// LS Electric XG5000 project: R11_plc
// PLC LoadWizard_PLC
// module base 0 slot 0: FEnet:XGL-EFMT(B) (Fast Ethernet Module, Electrical Master)
// module base 0 slot 1: Input Module:XGI-D24A/B (DC 24V Input, 32 Contacts)
// module base 0 slot 2: Output Module:XGQ-TR4A/B (Transistor Output, 32 Contacts (0.1A, Sink Output/Source Output))
// module base 0 slot 3: 64points reservation:XG-IN64

PROGRAM Main (task: Scan Program)

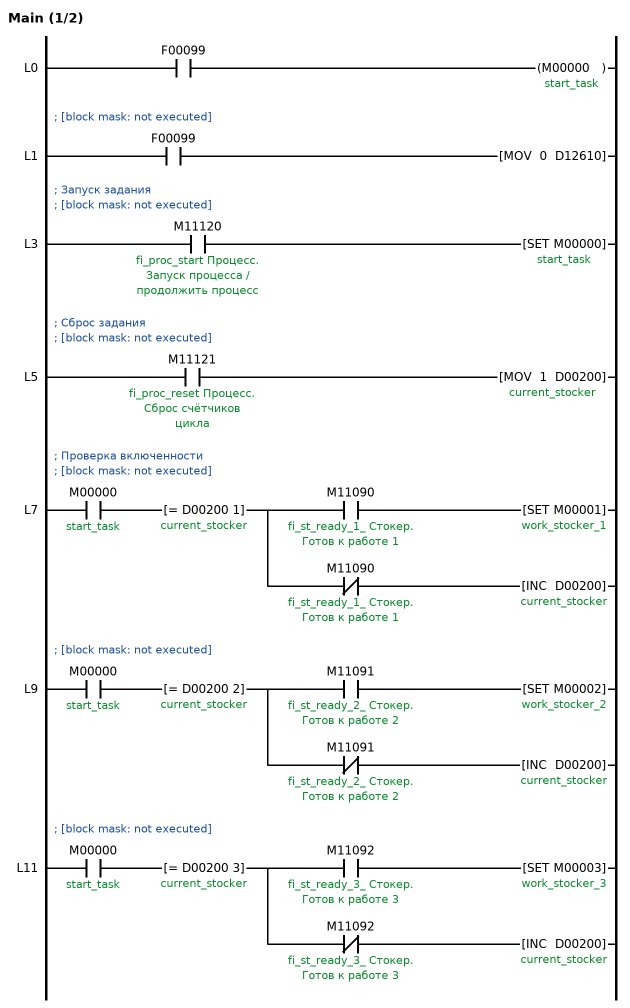
; L0
LOAD      F00099
OUT       M00000	// start_task
; L1 (block mask: not executed)
LOAD      F00099
MOV       0 D12610
// Запуск задания
; L3 (block mask: not executed)
LOAD      M11120	// fi_proc_start Процесс. Запуск процесса / продолжить процесс
SET       M00000	// start_task
// Сброс задания
; L5 (block mask: not executed)
LOAD      M11121	// fi_proc_reset Процесс. Сброс счётчиков цикла
MOV       1 D00200	// current_stocker
// Проверка включенности
; L7 (block mask: not executed)
LOAD      M00000	// start_task
AND=      D00200 1	// current_stocker
MPUSH
AND       M11090	// fi_st_ready_1_ Стокер. Готов к работе 1
SET       M00001	// work_stocker_1
MPOP
AND NOT   M11090	// fi_st_ready_1_ Стокер. Готов к работе 1
INC       D00200	// current_stocker
; L9 (block mask: not executed)
LOAD      M00000	// start_task
AND=      D00200 2	// current_stocker
MPUSH
AND       M11091	// fi_st_ready_2_ Стокер. Готов к работе 2
SET       M00002	// work_stocker_2
MPOP
AND NOT   M11091	// fi_st_ready_2_ Стокер. Готов к работе 2
INC       D00200	// current_stocker
; L11 (block mask: not executed)
LOAD      M00000	// start_task
AND=      D00200 3	// current_stocker
MPUSH
AND       M11092	// fi_st_ready_3_ Стокер. Готов к работе 3
SET       M00003	// work_stocker_3
MPOP
AND NOT   M11092	// fi_st_ready_3_ Стокер. Готов к работе 3
INC       D00200	// current_stocker

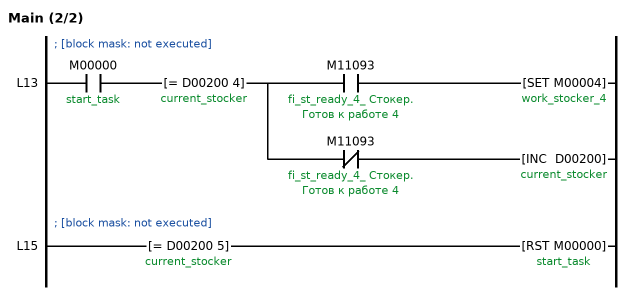
; L13 (block mask: not executed)
LOAD      M00000	// start_task
AND=      D00200 4	// current_stocker
MPUSH
AND       M11093	// fi_st_ready_4_ Стокер. Готов к работе 4
SET       M00004	// work_stocker_4
MPOP
AND NOT   M11093	// fi_st_ready_4_ Стокер. Готов к работе 4
INC       D00200	// current_stocker
; L15 (block mask: not executed)
LOAD=     D00200 5	// current_stocker
RST       M00000	// start_task

PROGRAM CNC (task: Scan Program)

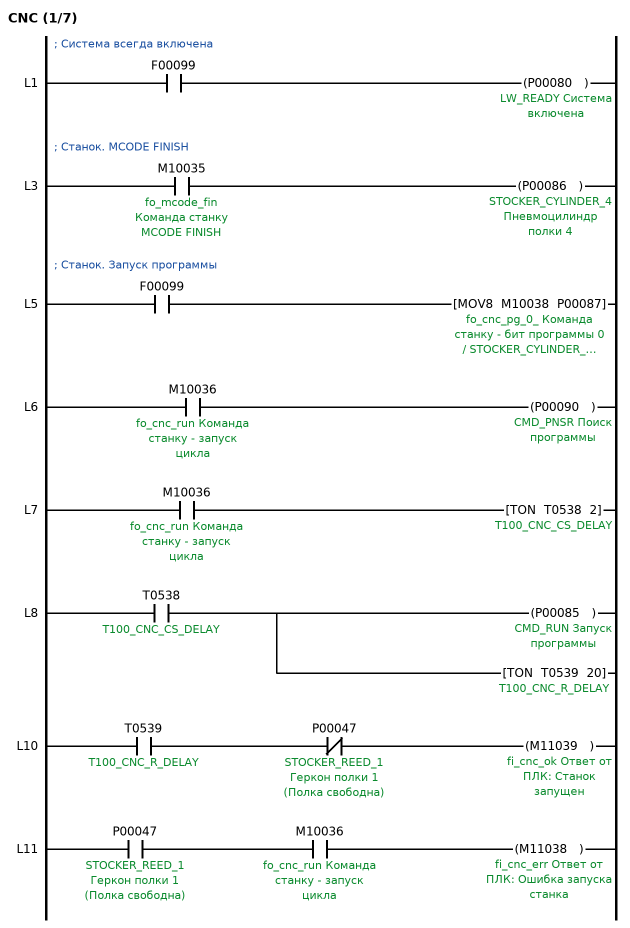
// Система всегда включена
; L1
LOAD      F00099
OUT       P00080	// LW_READY Система включена
// Станок. MCODE FINISH
; L3
LOAD      M10035	// fo_mcode_fin Команда станку  MCODE FINISH
OUT       P00086	// STOCKER_CYLINDER_4 Пневмоцилиндр полки 4
// Станок. Запуск программы
; L5
LOAD      F00099
MOV8      M10038 P00087	// fo_cnc_pg_0_ Команда станку - бит программы 0 / STOCKER_CYLINDER_3 Пневмоцилиндр полки 3
; L6
LOAD      M10036	// fo_cnc_run Команда станку - запуск цикла
OUT       P00090	// CMD_PNSR Поиск программы
; L7
LOAD      M10036	// fo_cnc_run Команда станку - запуск цикла
TON       T0538 2	// T100_CNC_CS_DELAY
; L8
LOAD      T0538	// T100_CNC_CS_DELAY
OUT       P00085	// CMD_RUN Запуск программы
TON       T0539 20	// T100_CNC_R_DELAY
; L10
LOAD      T0539	// T100_CNC_R_DELAY
AND NOT   P00047	// STOCKER_REED_1 Геркон полки 1 (Полка свободна)
OUT       M11039	// fi_cnc_ok Ответ от ПЛК: Станок запущен 
; L11
LOAD      P00047	// STOCKER_REED_1 Геркон полки 1 (Полка свободна)
AND       M10036	// fo_cnc_run Команда станку - запуск цикла
OUT       M11038	// fi_cnc_err Ответ от ПЛК: Ошибка запуска станка

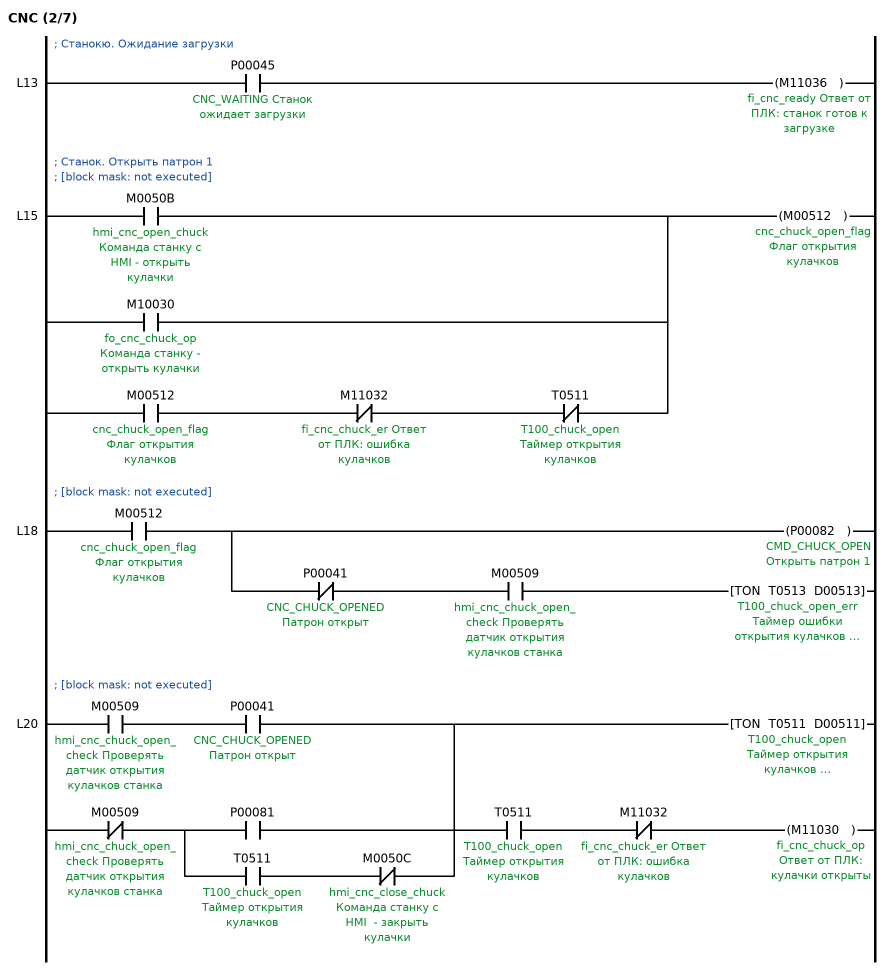
// Станокю. Ожидание загрузки
; L13
LOAD      P00045	// CNC_WAITING Станок ожидает загрузки
OUT       M11036	// fi_cnc_ready Ответ от ПЛК: станок готов к загрузке
// Станок. Открыть патрон 1
; L15 (block mask: not executed)
LOAD      M0050B	// hmi_cnc_open_chuck Команда станку с HMI - открыть кулачки
OR        M10030	// fo_cnc_chuck_op Команда станку - открыть кулачки
LOAD      M00512	// cnc_chuck_open_flag Флаг открытия кулачков
AND NOT   M11032	// fi_cnc_chuck_er Ответ от ПЛК: ошибка кулачков
AND NOT   T0511	// T100_chuck_open Таймер открытия кулачков
OR LOAD
OUT       M00512	// cnc_chuck_open_flag Флаг открытия кулачков
; L18 (block mask: not executed)
LOAD      M00512	// cnc_chuck_open_flag Флаг открытия кулачков
OUT       P00082	// CMD_CHUCK_OPEN Открыть патрон 1
AND NOT   P00041	// CNC_CHUCK_OPENED Патрон открыт
AND       M00509	// hmi_cnc_chuck_open_check Проверять датчик открытия кулачков станка
TON       T0513 D00513	// T100_chuck_open_err Таймер ошибки открытия кулачков / hmi_chuck_err_time Время ошибки кулачков
; L20 (block mask: not executed)
LOAD      M00509	// hmi_cnc_chuck_open_check Проверять датчик открытия кулачков станка
AND       P00041	// CNC_CHUCK_OPENED Патрон открыт
LOAD NOT  M00509	// hmi_cnc_chuck_open_check Проверять датчик открытия кулачков станка
LOAD      P00081
LOAD      T0511	// T100_chuck_open Таймер открытия кулачков
AND NOT   M0050C	// hmi_cnc_close_chuck Команда станку с HMI  - закрыть кулачки
OR LOAD
AND LOAD
OR LOAD
TON       T0511 D00511	// T100_chuck_open Таймер открытия кулачков / hmi_chuck_open_time Время на открытие кулачков
AND       T0511	// T100_chuck_open Таймер открытия кулачков
AND NOT   M11032	// fi_cnc_chuck_er Ответ от ПЛК: ошибка кулачков
OUT       M11030	// fi_cnc_chuck_op Ответ от ПЛК: кулачки открыты

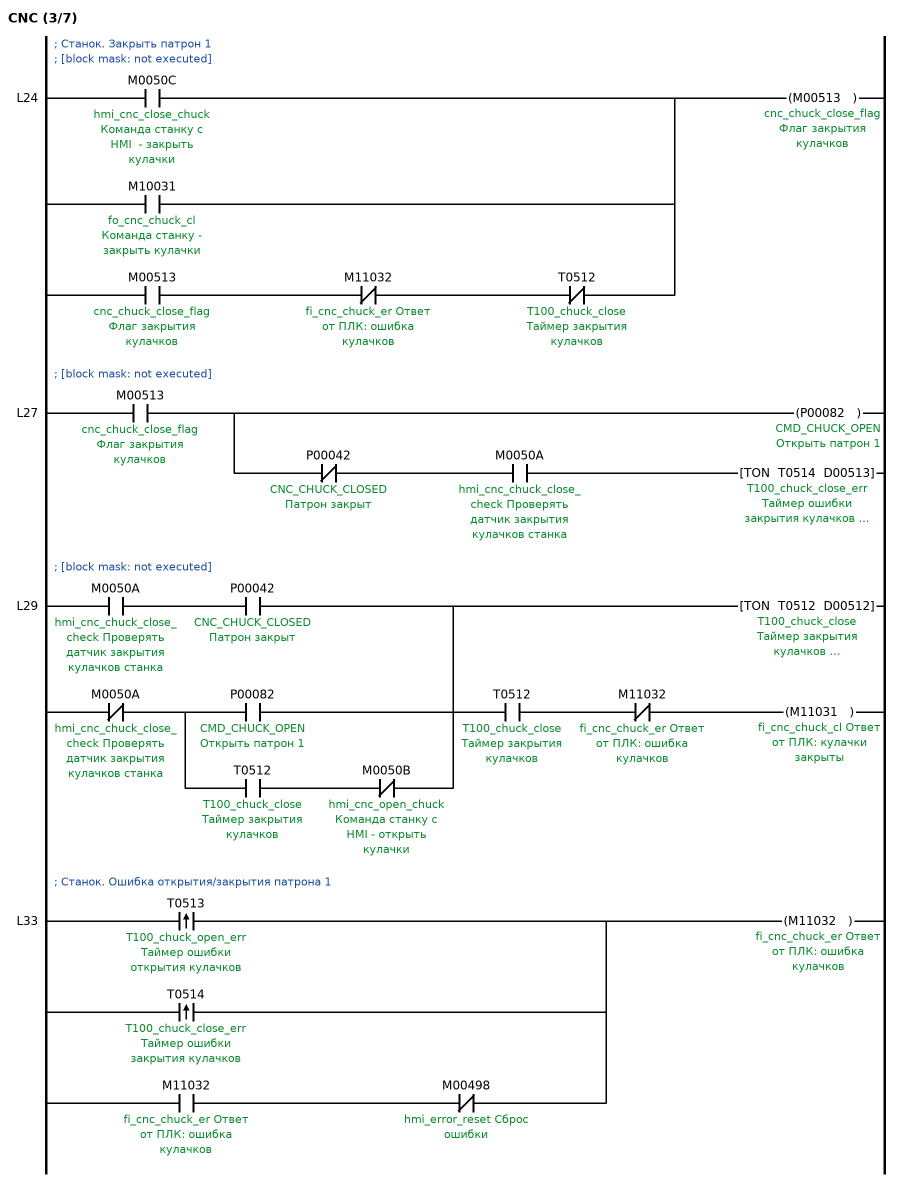
// Станок. Закрыть патрон 1
; L24 (block mask: not executed)
LOAD      M0050C	// hmi_cnc_close_chuck Команда станку с HMI  - закрыть кулачки
OR        M10031	// fo_cnc_chuck_cl Команда станку - закрыть кулачки
LOAD      M00513	// cnc_chuck_close_flag Флаг закрытия кулачков
AND NOT   M11032	// fi_cnc_chuck_er Ответ от ПЛК: ошибка кулачков
AND NOT   T0512	// T100_chuck_close Таймер закрытия кулачков
OR LOAD
OUT       M00513	// cnc_chuck_close_flag Флаг закрытия кулачков
; L27 (block mask: not executed)
LOAD      M00513	// cnc_chuck_close_flag Флаг закрытия кулачков
OUT       P00082	// CMD_CHUCK_OPEN Открыть патрон 1
AND NOT   P00042	// CNC_CHUCK_CLOSED Патрон закрыт
AND       M0050A	// hmi_cnc_chuck_close_check Проверять датчик закрытия кулачков станка
TON       T0514 D00513	// T100_chuck_close_err Таймер ошибки закрытия кулачков / hmi_chuck_err_time Время ошибки кулачков
; L29 (block mask: not executed)
LOAD      M0050A	// hmi_cnc_chuck_close_check Проверять датчик закрытия кулачков станка
AND       P00042	// CNC_CHUCK_CLOSED Патрон закрыт
LOAD NOT  M0050A	// hmi_cnc_chuck_close_check Проверять датчик закрытия кулачков станка
LOAD      P00082	// CMD_CHUCK_OPEN Открыть патрон 1
LOAD      T0512	// T100_chuck_close Таймер закрытия кулачков
AND NOT   M0050B	// hmi_cnc_open_chuck Команда станку с HMI - открыть кулачки
OR LOAD
AND LOAD
OR LOAD
TON       T0512 D00512	// T100_chuck_close Таймер закрытия кулачков / hmi_chuck_close_time Время на закрытие кулачков
AND       T0512	// T100_chuck_close Таймер закрытия кулачков
AND NOT   M11032	// fi_cnc_chuck_er Ответ от ПЛК: ошибка кулачков
OUT       M11031	// fi_cnc_chuck_cl Ответ от ПЛК: кулачки закрыты
// Станок. Ошибка открытия/закрытия патрона 1
; L33
LOADP     T0513	// T100_chuck_open_err Таймер ошибки открытия кулачков
ORP       T0514	// T100_chuck_close_err Таймер ошибки закрытия кулачков
LOAD      M11032	// fi_cnc_chuck_er Ответ от ПЛК: ошибка кулачков
AND NOT   M00498	// hmi_error_reset Сброс ошибки
OR LOAD
OUT       M11032	// fi_cnc_chuck_er Ответ от ПЛК: ошибка кулачков

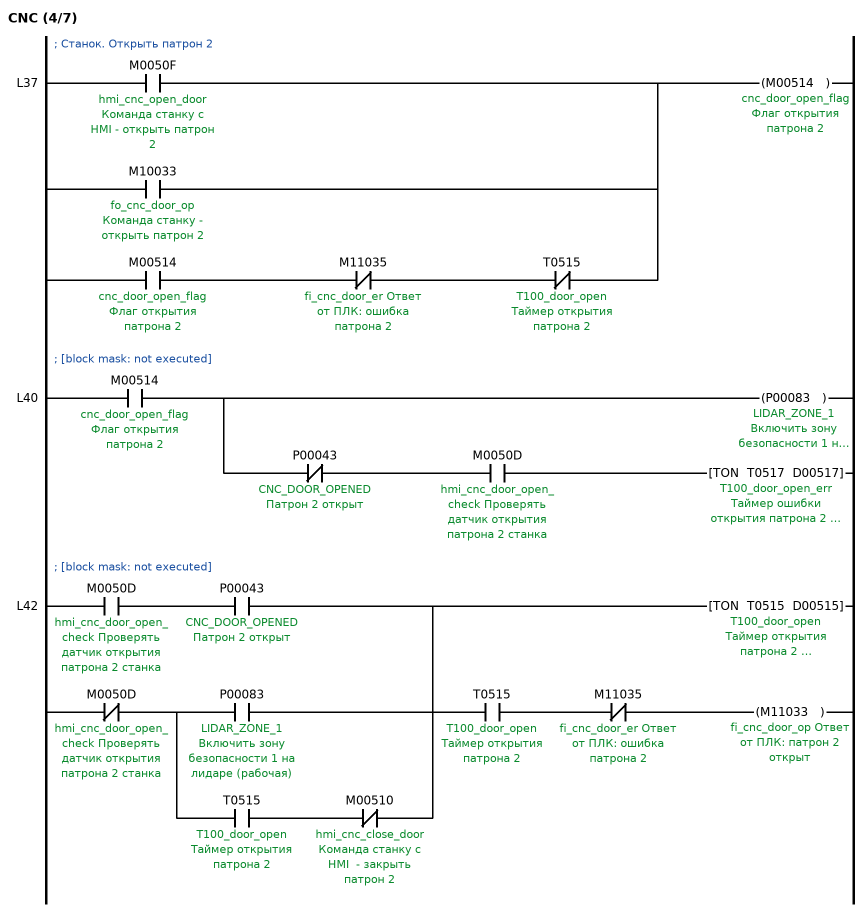
// Станок. Открыть патрон 2
; L37
LOAD      M0050F	// hmi_cnc_open_door Команда станку с HMI - открыть патрон 2
OR        M10033	// fo_cnc_door_op Команда станку - открыть патрон 2
LOAD      M00514	// cnc_door_open_flag Флаг открытия патрона 2
AND NOT   M11035	// fi_cnc_door_er Ответ от ПЛК: ошибка патрона 2
AND NOT   T0515	// T100_door_open Таймер открытия патрона 2
OR LOAD
OUT       M00514	// cnc_door_open_flag Флаг открытия патрона 2
; L40 (block mask: not executed)
LOAD      M00514	// cnc_door_open_flag Флаг открытия патрона 2
OUT       P00083	// LIDAR_ZONE_1 Включить зону безопасности 1 на лидаре (рабочая)
AND NOT   P00043	// CNC_DOOR_OPENED Патрон 2 открыт
AND       M0050D	// hmi_cnc_door_open_check Проверять датчик открытия патрона 2 станка
TON       T0517 D00517	// T100_door_open_err Таймер ошибки открытия патрона 2 / hmi_door_err_time Время ошибки патрона 2
; L42 (block mask: not executed)
LOAD      M0050D	// hmi_cnc_door_open_check Проверять датчик открытия патрона 2 станка
AND       P00043	// CNC_DOOR_OPENED Патрон 2 открыт
LOAD NOT  M0050D	// hmi_cnc_door_open_check Проверять датчик открытия патрона 2 станка
LOAD      P00083	// LIDAR_ZONE_1 Включить зону безопасности 1 на лидаре (рабочая)
LOAD      T0515	// T100_door_open Таймер открытия патрона 2
AND NOT   M00510	// hmi_cnc_close_door Команда станку с HMI  - закрыть патрон 2
OR LOAD
AND LOAD
OR LOAD
TON       T0515 D00515	// T100_door_open Таймер открытия патрона 2 / hmi_door_open_time Время на открытие патрона 2
AND       T0515	// T100_door_open Таймер открытия патрона 2
AND NOT   M11035	// fi_cnc_door_er Ответ от ПЛК: ошибка патрона 2
OUT       M11033	// fi_cnc_door_op Ответ от ПЛК: патрон 2 открыт

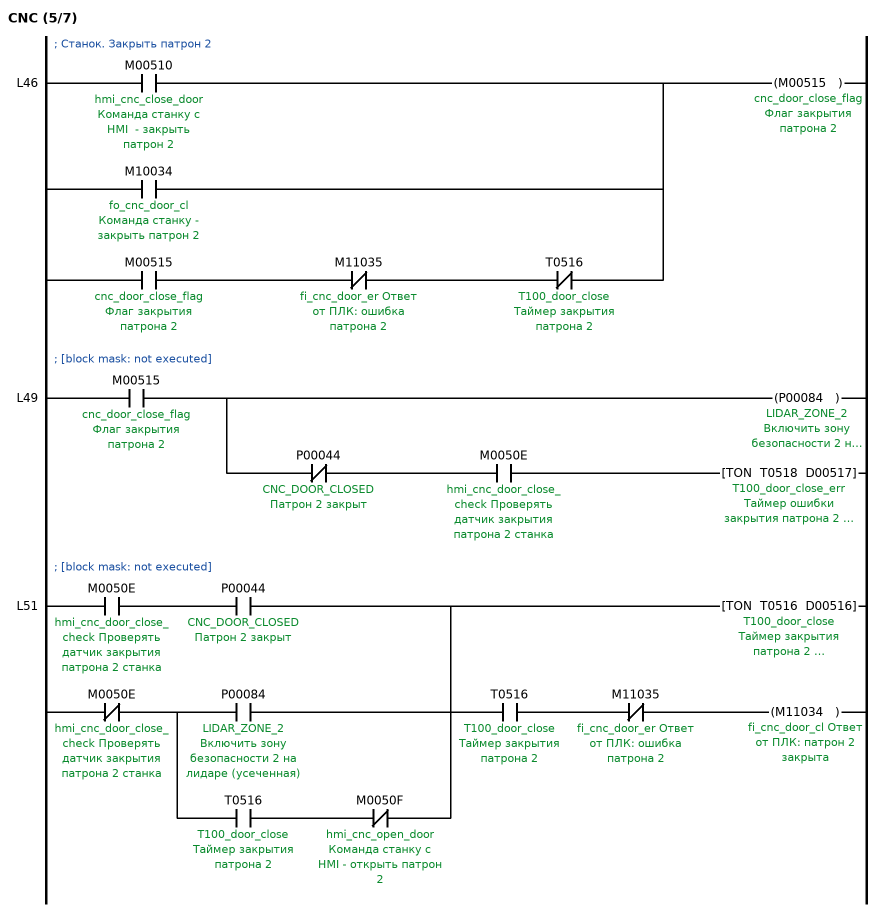
// Станок. Закрыть патрон 2
; L46
LOAD      M00510	// hmi_cnc_close_door Команда станку с HMI  - закрыть патрон 2
OR        M10034	// fo_cnc_door_cl Команда станку - закрыть патрон 2
LOAD      M00515	// cnc_door_close_flag Флаг закрытия патрона 2
AND NOT   M11035	// fi_cnc_door_er Ответ от ПЛК: ошибка патрона 2
AND NOT   T0516	// T100_door_close Таймер закрытия патрона 2
OR LOAD
OUT       M00515	// cnc_door_close_flag Флаг закрытия патрона 2
; L49 (block mask: not executed)
LOAD      M00515	// cnc_door_close_flag Флаг закрытия патрона 2
OUT       P00084	// LIDAR_ZONE_2 Включить зону безопасности 2 на лидаре (усеченная)
AND NOT   P00044	// CNC_DOOR_CLOSED Патрон 2 закрыт
AND       M0050E	// hmi_cnc_door_close_check Проверять датчик закрытия патрона 2 станка
TON       T0518 D00517	// T100_door_close_err Таймер ошибки закрытия патрона 2 / hmi_door_err_time Время ошибки патрона 2
; L51 (block mask: not executed)
LOAD      M0050E	// hmi_cnc_door_close_check Проверять датчик закрытия патрона 2 станка
AND       P00044	// CNC_DOOR_CLOSED Патрон 2 закрыт
LOAD NOT  M0050E	// hmi_cnc_door_close_check Проверять датчик закрытия патрона 2 станка
LOAD      P00084	// LIDAR_ZONE_2 Включить зону безопасности 2 на лидаре (усеченная)
LOAD      T0516	// T100_door_close Таймер закрытия патрона 2
AND NOT   M0050F	// hmi_cnc_open_door Команда станку с HMI - открыть патрон 2
OR LOAD
AND LOAD
OR LOAD
TON       T0516 D00516	// T100_door_close Таймер закрытия патрона 2 / hmi_door_close_time Время на закрытие патрона 2
AND       T0516	// T100_door_close Таймер закрытия патрона 2
AND NOT   M11035	// fi_cnc_door_er Ответ от ПЛК: ошибка патрона 2
OUT       M11034	// fi_cnc_door_cl Ответ от ПЛК: патрон 2 закрыта

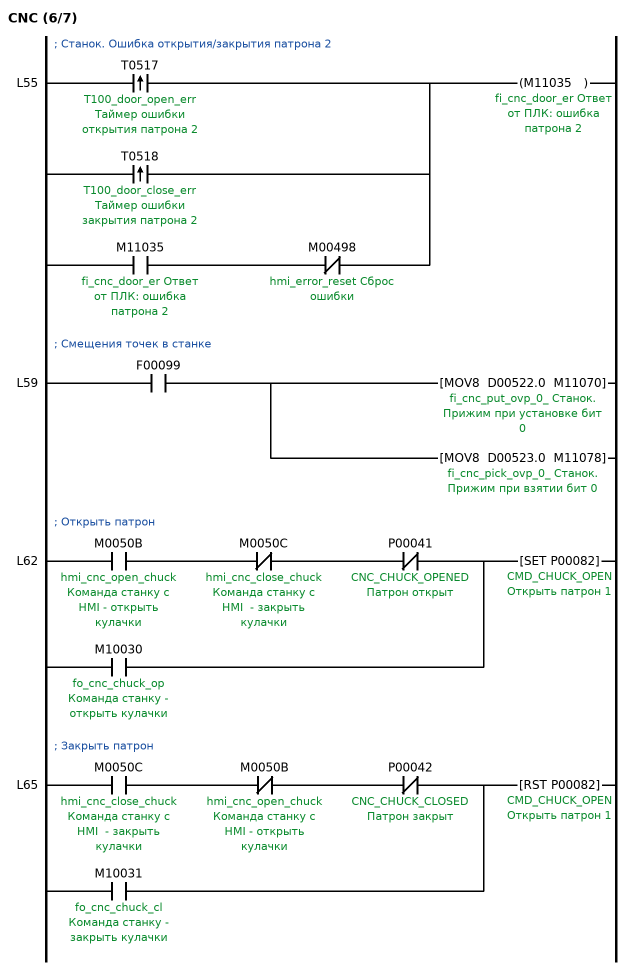
// Станок. Ошибка открытия/закрытия патрона 2
; L55
LOADP     T0517	// T100_door_open_err Таймер ошибки открытия патрона 2
ORP       T0518	// T100_door_close_err Таймер ошибки закрытия патрона 2
LOAD      M11035	// fi_cnc_door_er Ответ от ПЛК: ошибка патрона 2
AND NOT   M00498	// hmi_error_reset Сброс ошибки
OR LOAD
OUT       M11035	// fi_cnc_door_er Ответ от ПЛК: ошибка патрона 2
// Смещения точек в станке
; L59
LOAD      F00099
MOV8      D00522.0 M11070	// fi_cnc_put_ovp_0_ Станок. Прижим при установке бит 0
MOV8      D00523.0 M11078	// fi_cnc_pick_ovp_0_ Станок. Прижим при взятии бит 0
// Открыть патрон
; L62
LOAD      M0050B	// hmi_cnc_open_chuck Команда станку с HMI - открыть кулачки
AND NOT   M0050C	// hmi_cnc_close_chuck Команда станку с HMI  - закрыть кулачки
AND NOT   P00041	// CNC_CHUCK_OPENED Патрон открыт
OR        M10030	// fo_cnc_chuck_op Команда станку - открыть кулачки
SET       P00082	// CMD_CHUCK_OPEN Открыть патрон 1
// Закрыть патрон
; L65
LOAD      M0050C	// hmi_cnc_close_chuck Команда станку с HMI  - закрыть кулачки
AND NOT   M0050B	// hmi_cnc_open_chuck Команда станку с HMI - открыть кулачки
AND NOT   P00042	// CNC_CHUCK_CLOSED Патрон закрыт
OR        M10031	// fo_cnc_chuck_cl Команда станку - закрыть кулачки
RST       P00082	// CMD_CHUCK_OPEN Открыть патрон 1

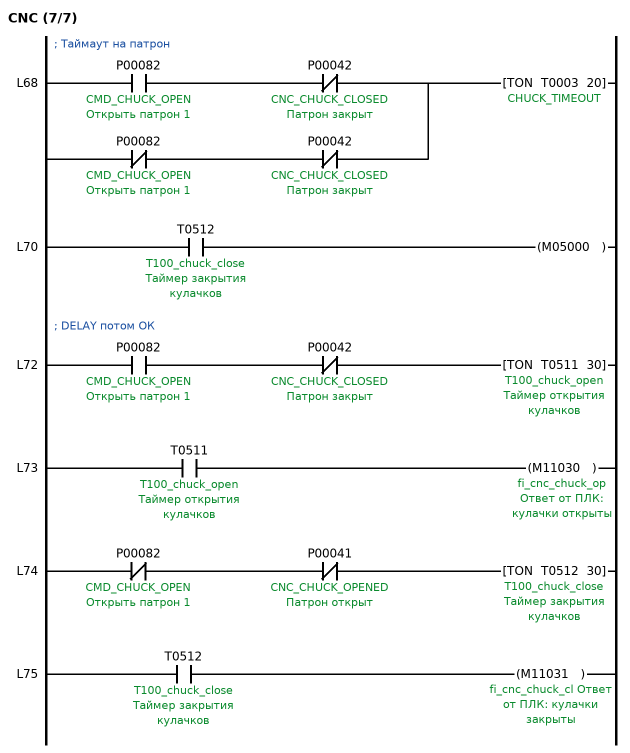
// Таймаут на патрон
; L68
LOAD      P00082	// CMD_CHUCK_OPEN Открыть патрон 1
AND NOT   P00042	// CNC_CHUCK_CLOSED Патрон закрыт
LOAD NOT  P00082	// CMD_CHUCK_OPEN Открыть патрон 1
AND NOT   P00042	// CNC_CHUCK_CLOSED Патрон закрыт
OR LOAD
TON       T0003 20	// CHUCK_TIMEOUT
; L70
LOAD      T0512	// T100_chuck_close Таймер закрытия кулачков
OUT       M05000
// DELAY потом ОК
; L72
LOAD      P00082	// CMD_CHUCK_OPEN Открыть патрон 1
AND NOT   P00042	// CNC_CHUCK_CLOSED Патрон закрыт
TON       T0511 30	// T100_chuck_open Таймер открытия кулачков
; L73
LOAD      T0511	// T100_chuck_open Таймер открытия кулачков
OUT       M11030	// fi_cnc_chuck_op Ответ от ПЛК: кулачки открыты
; L74
LOAD NOT  P00082	// CMD_CHUCK_OPEN Открыть патрон 1
AND NOT   P00041	// CNC_CHUCK_OPENED Патрон открыт
TON       T0512 30	// T100_chuck_close Таймер закрытия кулачков
; L75
LOAD      T0512	// T100_chuck_close Таймер закрытия кулачков
OUT       M11031	// fi_cnc_chuck_cl Ответ от ПЛК: кулачки закрыты

PROGRAM STOCKER (task: Scan Program)

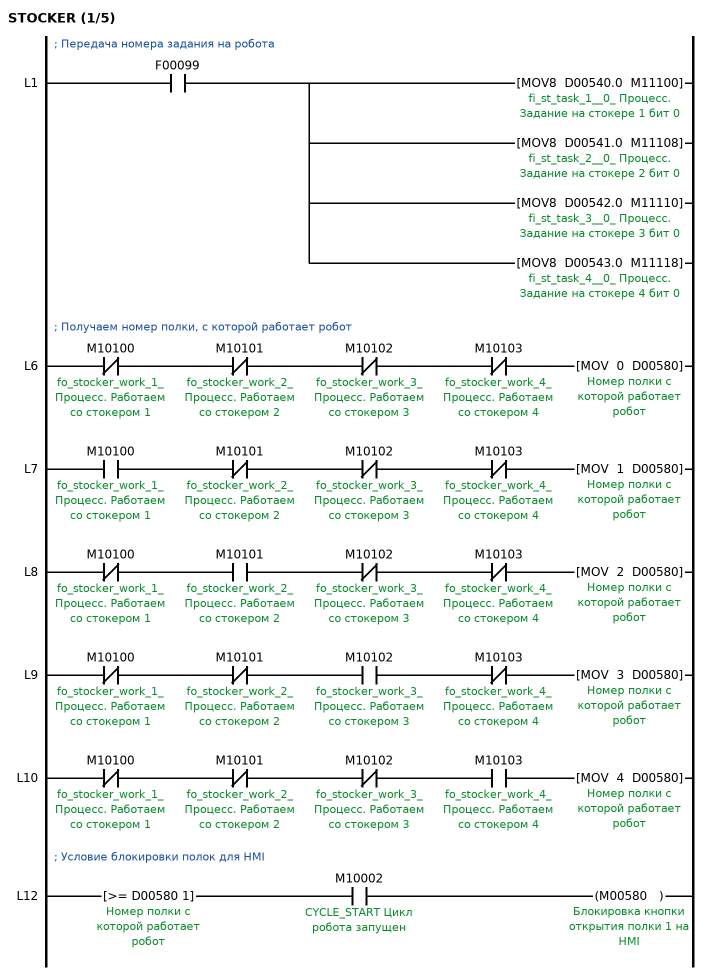
// Передача номера задания на робота
; L1
LOAD      F00099
MOV8      D00540.0 M11100	// fi_st_task_1__0_ Процесс. Задание на стокере 1 бит 0
MOV8      D00541.0 M11108	// fi_st_task_2__0_ Процесс. Задание на стокере 2 бит 0
MOV8      D00542.0 M11110	// fi_st_task_3__0_ Процесс. Задание на стокере 3 бит 0
MOV8      D00543.0 M11118	// fi_st_task_4__0_ Процесс. Задание на стокере 4 бит 0
// Получаем номер полки, с которой работает робот
; L6
LOAD NOT  M10100	// fo_stocker_work_1_ Процесс. Работаем со стокером 1
AND NOT   M10101	// fo_stocker_work_2_ Процесс. Работаем со стокером 2
AND NOT   M10102	// fo_stocker_work_3_ Процесс. Работаем со стокером 3
AND NOT   M10103	// fo_stocker_work_4_ Процесс. Работаем со стокером 4
MOV       0 D00580	// Номер полки с которой работает робот
; L7
LOAD      M10100	// fo_stocker_work_1_ Процесс. Работаем со стокером 1
AND NOT   M10101	// fo_stocker_work_2_ Процесс. Работаем со стокером 2
AND NOT   M10102	// fo_stocker_work_3_ Процесс. Работаем со стокером 3
AND NOT   M10103	// fo_stocker_work_4_ Процесс. Работаем со стокером 4
MOV       1 D00580	// Номер полки с которой работает робот
; L8
LOAD NOT  M10100	// fo_stocker_work_1_ Процесс. Работаем со стокером 1
AND       M10101	// fo_stocker_work_2_ Процесс. Работаем со стокером 2
AND NOT   M10102	// fo_stocker_work_3_ Процесс. Работаем со стокером 3
AND NOT   M10103	// fo_stocker_work_4_ Процесс. Работаем со стокером 4
MOV       2 D00580	// Номер полки с которой работает робот
; L9
LOAD NOT  M10100	// fo_stocker_work_1_ Процесс. Работаем со стокером 1
AND NOT   M10101	// fo_stocker_work_2_ Процесс. Работаем со стокером 2
AND       M10102	// fo_stocker_work_3_ Процесс. Работаем со стокером 3
AND NOT   M10103	// fo_stocker_work_4_ Процесс. Работаем со стокером 4
MOV       3 D00580	// Номер полки с которой работает робот
; L10
LOAD NOT  M10100	// fo_stocker_work_1_ Процесс. Работаем со стокером 1
AND NOT   M10101	// fo_stocker_work_2_ Процесс. Работаем со стокером 2
AND NOT   M10102	// fo_stocker_work_3_ Процесс. Работаем со стокером 3
AND       M10103	// fo_stocker_work_4_ Процесс. Работаем со стокером 4
MOV       4 D00580	// Номер полки с которой работает робот
// Условие блокировки полок для HMI
; L12
LOAD>=    D00580 1	// Номер полки с которой работает робот
AND       M10002	// CYCLE_START Цикл робота запущен
OUT       M00580	// Блокировка кнопки открытия полки 1 на HMI

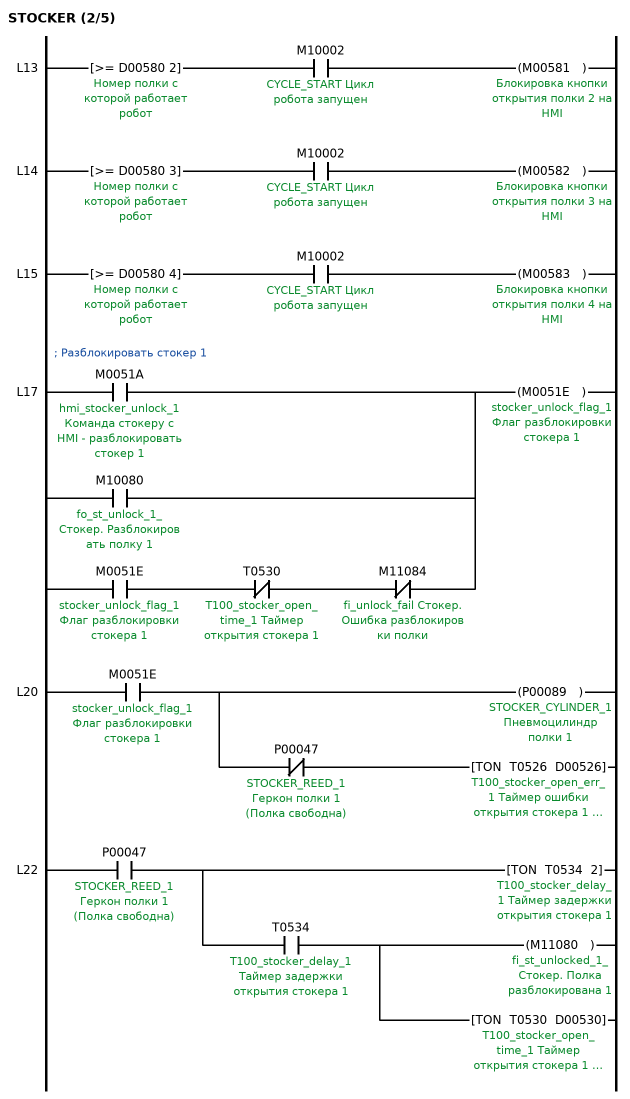
; L13
LOAD>=    D00580 2	// Номер полки с которой работает робот
AND       M10002	// CYCLE_START Цикл робота запущен
OUT       M00581	// Блокировка кнопки открытия полки 2 на HMI
; L14
LOAD>=    D00580 3	// Номер полки с которой работает робот
AND       M10002	// CYCLE_START Цикл робота запущен
OUT       M00582	// Блокировка кнопки открытия полки 3 на HMI
; L15
LOAD>=    D00580 4	// Номер полки с которой работает робот
AND       M10002	// CYCLE_START Цикл робота запущен
OUT       M00583	// Блокировка кнопки открытия полки 4 на HMI
// Разблокировать стокер 1
; L17
LOAD      M0051A	// hmi_stocker_unlock_1 Команда стокеру с HMI - разблокировать стокер 1
OR        M10080	// fo_st_unlock_1_ Стокер. Разблокировать полку 1
LOAD      M0051E	// stocker_unlock_flag_1 Флаг разблокировки стокера 1
AND NOT   T0530	// T100_stocker_open_time_1 Таймер открытия стокера 1
AND NOT   M11084	// fi_unlock_fail Стокер. Ошибка разблокировки полки
OR LOAD
OUT       M0051E	// stocker_unlock_flag_1 Флаг разблокировки стокера 1
; L20
LOAD      M0051E	// stocker_unlock_flag_1 Флаг разблокировки стокера 1
OUT       P00089	// STOCKER_CYLINDER_1 Пневмоцилиндр полки 1
AND NOT   P00047	// STOCKER_REED_1 Геркон полки 1 (Полка свободна)
TON       T0526 D00526	// T100_stocker_open_err_1 Таймер ошибки открытия стокера 1 / hmi_stocker_err_time Время ошибки стокера
; L22
LOAD      P00047	// STOCKER_REED_1 Геркон полки 1 (Полка свободна)
TON       T0534 2	// T100_stocker_delay_1 Таймер задержки открытия стокера 1
AND       T0534	// T100_stocker_delay_1 Таймер задержки открытия стокера 1
OUT       M11080	// fi_st_unlocked_1_ Стокер. Полка разблокирована 1
TON       T0530 D00530	// T100_stocker_open_time_1 Таймер открытия стокера 1 / hmi_stocker_open_time Время открытия стокера 

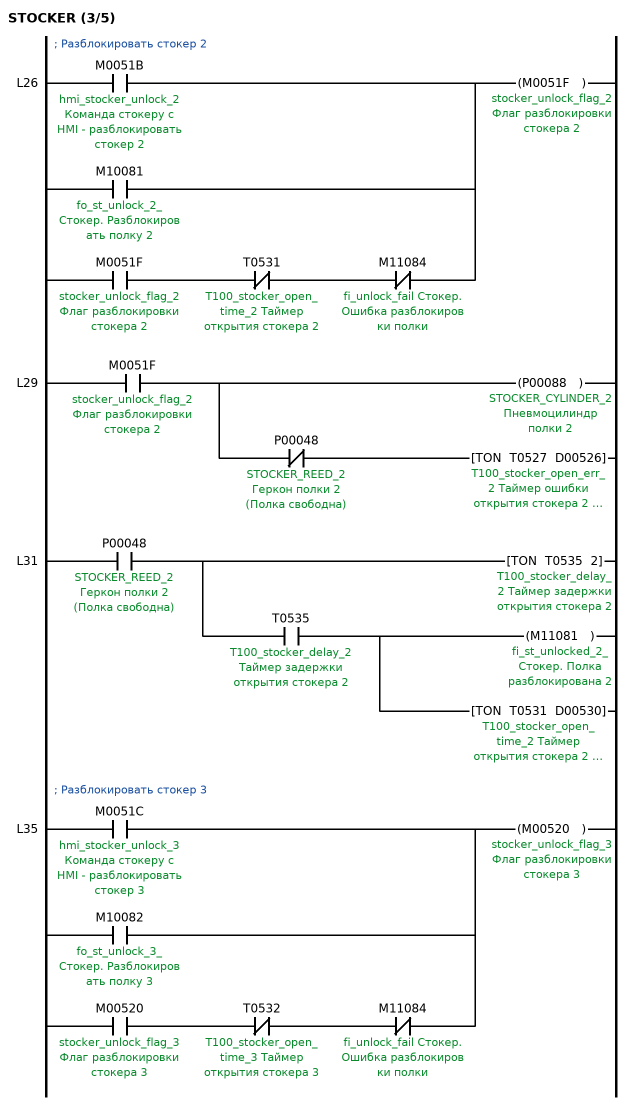
// Разблокировать стокер 2
; L26
LOAD      M0051B	// hmi_stocker_unlock_2 Команда стокеру с HMI - разблокировать стокер 2
OR        M10081	// fo_st_unlock_2_ Стокер. Разблокировать полку 2
LOAD      M0051F	// stocker_unlock_flag_2 Флаг разблокировки стокера 2
AND NOT   T0531	// T100_stocker_open_time_2 Таймер открытия стокера 2
AND NOT   M11084	// fi_unlock_fail Стокер. Ошибка разблокировки полки
OR LOAD
OUT       M0051F	// stocker_unlock_flag_2 Флаг разблокировки стокера 2
; L29
LOAD      M0051F	// stocker_unlock_flag_2 Флаг разблокировки стокера 2
OUT       P00088	// STOCKER_CYLINDER_2 Пневмоцилиндр полки 2
AND NOT   P00048	// STOCKER_REED_2 Геркон полки 2 (Полка свободна)
TON       T0527 D00526	// T100_stocker_open_err_2 Таймер ошибки открытия стокера 2 / hmi_stocker_err_time Время ошибки стокера
; L31
LOAD      P00048	// STOCKER_REED_2 Геркон полки 2 (Полка свободна)
TON       T0535 2	// T100_stocker_delay_2 Таймер задержки открытия стокера 2
AND       T0535	// T100_stocker_delay_2 Таймер задержки открытия стокера 2
OUT       M11081	// fi_st_unlocked_2_ Стокер. Полка разблокирована 2
TON       T0531 D00530	// T100_stocker_open_time_2 Таймер открытия стокера 2 / hmi_stocker_open_time Время открытия стокера 
// Разблокировать стокер 3
; L35
LOAD      M0051C	// hmi_stocker_unlock_3 Команда стокеру с HMI - разблокировать стокер 3
OR        M10082	// fo_st_unlock_3_ Стокер. Разблокировать полку 3
LOAD      M00520	// stocker_unlock_flag_3 Флаг разблокировки стокера 3
AND NOT   T0532	// T100_stocker_open_time_3 Таймер открытия стокера 3
AND NOT   M11084	// fi_unlock_fail Стокер. Ошибка разблокировки полки
OR LOAD
OUT       M00520	// stocker_unlock_flag_3 Флаг разблокировки стокера 3

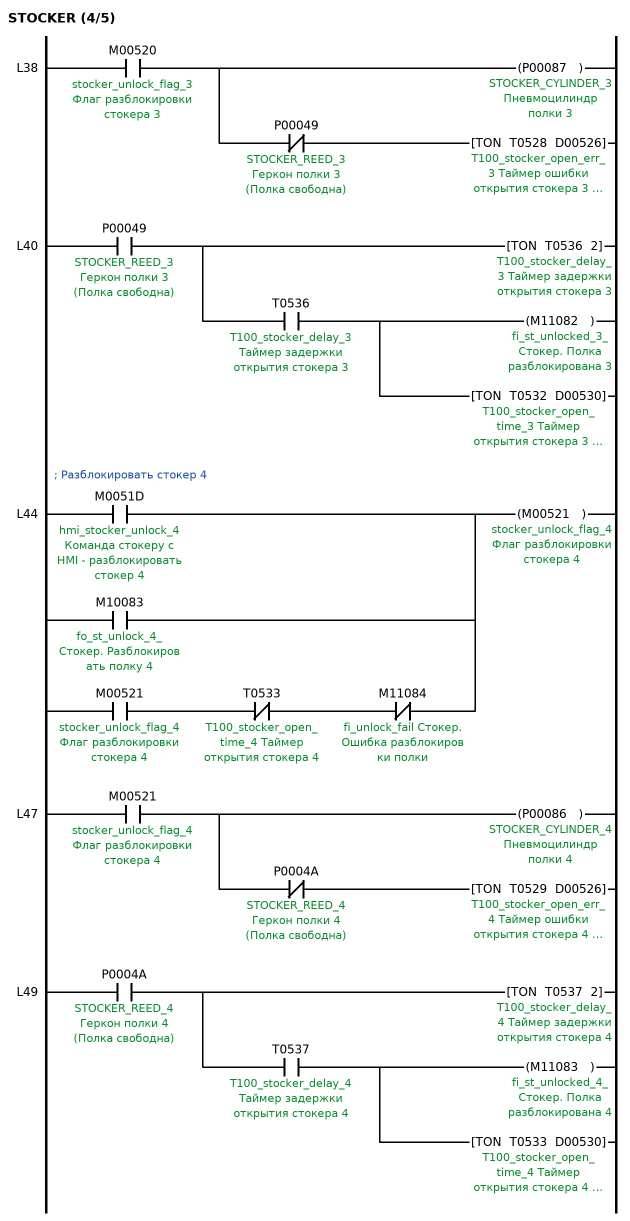
; L38
LOAD      M00520	// stocker_unlock_flag_3 Флаг разблокировки стокера 3
OUT       P00087	// STOCKER_CYLINDER_3 Пневмоцилиндр полки 3
AND NOT   P00049	// STOCKER_REED_3 Геркон полки 3 (Полка свободна)
TON       T0528 D00526	// T100_stocker_open_err_3 Таймер ошибки открытия стокера 3 / hmi_stocker_err_time Время ошибки стокера
; L40
LOAD      P00049	// STOCKER_REED_3 Геркон полки 3 (Полка свободна)
TON       T0536 2	// T100_stocker_delay_3 Таймер задержки открытия стокера 3
AND       T0536	// T100_stocker_delay_3 Таймер задержки открытия стокера 3
OUT       M11082	// fi_st_unlocked_3_ Стокер. Полка разблокирована 3
TON       T0532 D00530	// T100_stocker_open_time_3 Таймер открытия стокера 3 / hmi_stocker_open_time Время открытия стокера 
// Разблокировать стокер 4
; L44
LOAD      M0051D	// hmi_stocker_unlock_4 Команда стокеру с HMI - разблокировать стокер 4
OR        M10083	// fo_st_unlock_4_ Стокер. Разблокировать полку 4
LOAD      M00521	// stocker_unlock_flag_4 Флаг разблокировки стокера 4
AND NOT   T0533	// T100_stocker_open_time_4 Таймер открытия стокера 4
AND NOT   M11084	// fi_unlock_fail Стокер. Ошибка разблокировки полки
OR LOAD
OUT       M00521	// stocker_unlock_flag_4 Флаг разблокировки стокера 4
; L47
LOAD      M00521	// stocker_unlock_flag_4 Флаг разблокировки стокера 4
OUT       P00086	// STOCKER_CYLINDER_4 Пневмоцилиндр полки 4
AND NOT   P0004A	// STOCKER_REED_4 Геркон полки 4 (Полка свободна)
TON       T0529 D00526	// T100_stocker_open_err_4 Таймер ошибки открытия стокера 4 / hmi_stocker_err_time Время ошибки стокера
; L49
LOAD      P0004A	// STOCKER_REED_4 Геркон полки 4 (Полка свободна)
TON       T0537 2	// T100_stocker_delay_4 Таймер задержки открытия стокера 4
AND       T0537	// T100_stocker_delay_4 Таймер задержки открытия стокера 4
OUT       M11083	// fi_st_unlocked_4_ Стокер. Полка разблокирована 4
TON       T0533 D00530	// T100_stocker_open_time_4 Таймер открытия стокера 4 / hmi_stocker_open_time Время открытия стокера 

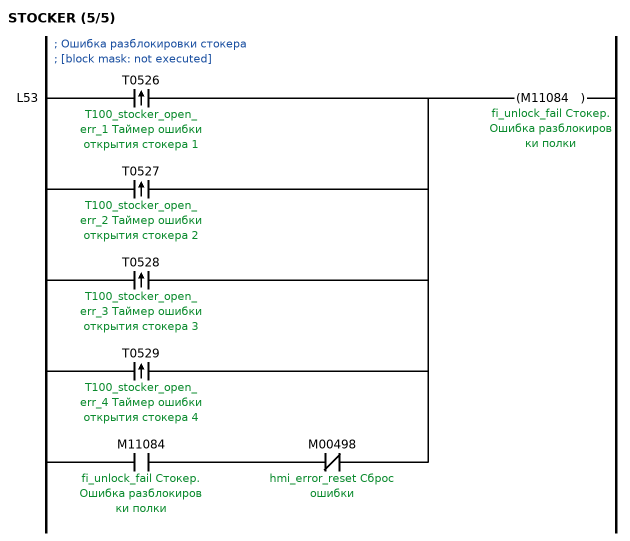
// Ошибка разблокировки стокера
; L53 (block mask: not executed)
LOADP     T0526	// T100_stocker_open_err_1 Таймер ошибки открытия стокера 1
ORP       T0527	// T100_stocker_open_err_2 Таймер ошибки открытия стокера 2
ORP       T0528	// T100_stocker_open_err_3 Таймер ошибки открытия стокера 3
ORP       T0529	// T100_stocker_open_err_4 Таймер ошибки открытия стокера 4
LOAD      M11084	// fi_unlock_fail Стокер. Ошибка разблокировки полки
AND NOT   M00498	// hmi_error_reset Сброс ошибки
OR LOAD
OUT       M11084	// fi_unlock_fail Стокер. Ошибка разблокировки полки

PROGRAM ROBOT (task: Scan Program)

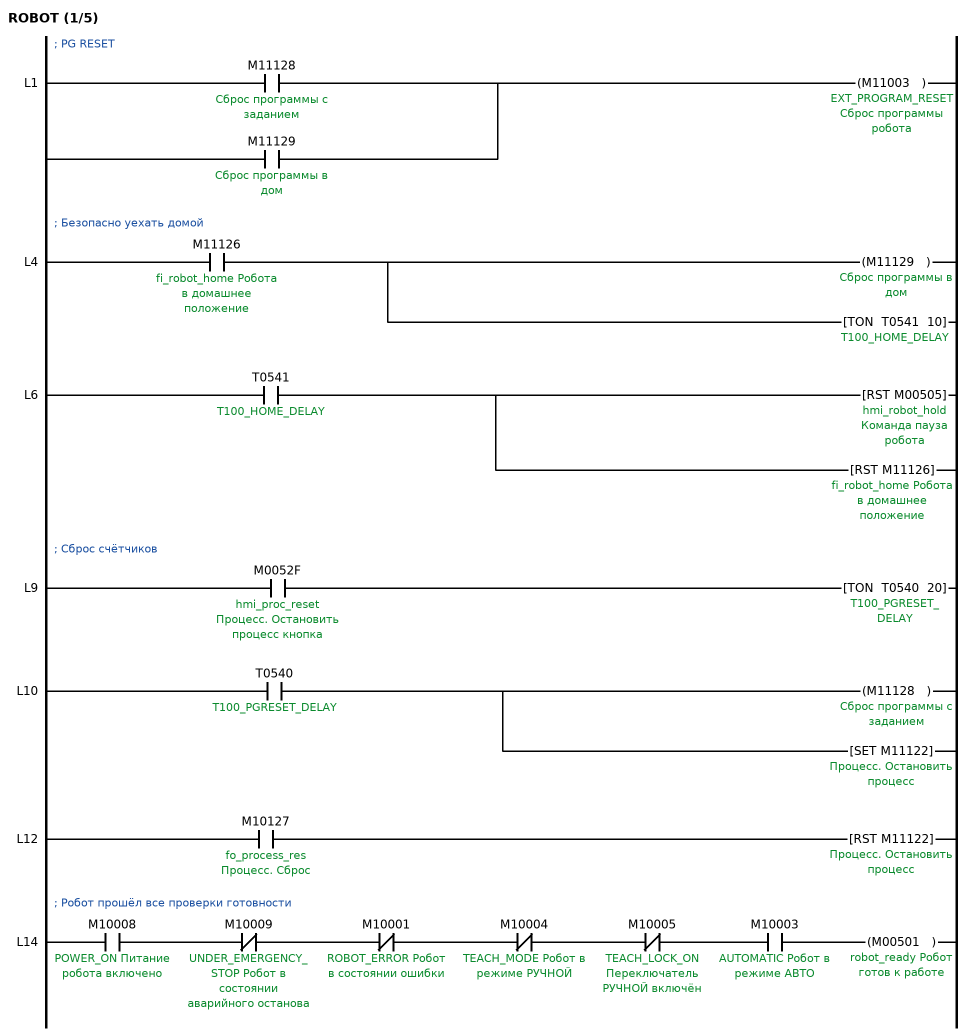
// PG RESET
; L1
LOAD      M11128	// Сброс программы с заданием
OR        M11129	// Сброс программы в дом
OUT       M11003	// EXT_PROGRAM_RESET Сброс программы робота
// Безопасно уехать домой
; L4
LOAD      M11126	// fi_robot_home Робота в домашнее положение
OUT       M11129	// Сброс программы в дом
TON       T0541 10	// T100_HOME_DELAY
; L6
LOAD      T0541	// T100_HOME_DELAY
RST       M00505	// hmi_robot_hold Команда пауза робота
RST       M11126	// fi_robot_home Робота в домашнее положение
// Сброс счётчиков
; L9
LOAD      M0052F	// hmi_proc_reset Процесс. Остановить процесс кнопка 
TON       T0540 20	// T100_PGRESET_DELAY
; L10
LOAD      T0540	// T100_PGRESET_DELAY
OUT       M11128	// Сброс программы с заданием
SET       M11122	// Процесс. Остановить процесс
; L12
LOAD      M10127	// fo_process_res Процесс. Сброс 
RST       M11122	// Процесс. Остановить процесс
// Робот прошёл все проверки готовности
; L14
LOAD      M10008	// POWER_ON Питание робота включено
AND NOT   M10009	// UNDER_EMERGENCY_STOP Робот в состоянии аварийного останова
AND NOT   M10001	// ROBOT_ERROR Робот в состоянии ошибки
AND NOT   M10004	// TEACH_MODE Робот в режиме РУЧНОЙ
AND NOT   M10005	// TEACH_LOCK_ON Переключатель РУЧНОЙ включён
AND       M10003	// AUTOMATIC Робот в режиме АВТО
OUT       M00501	// robot_ready Робот готов к работе

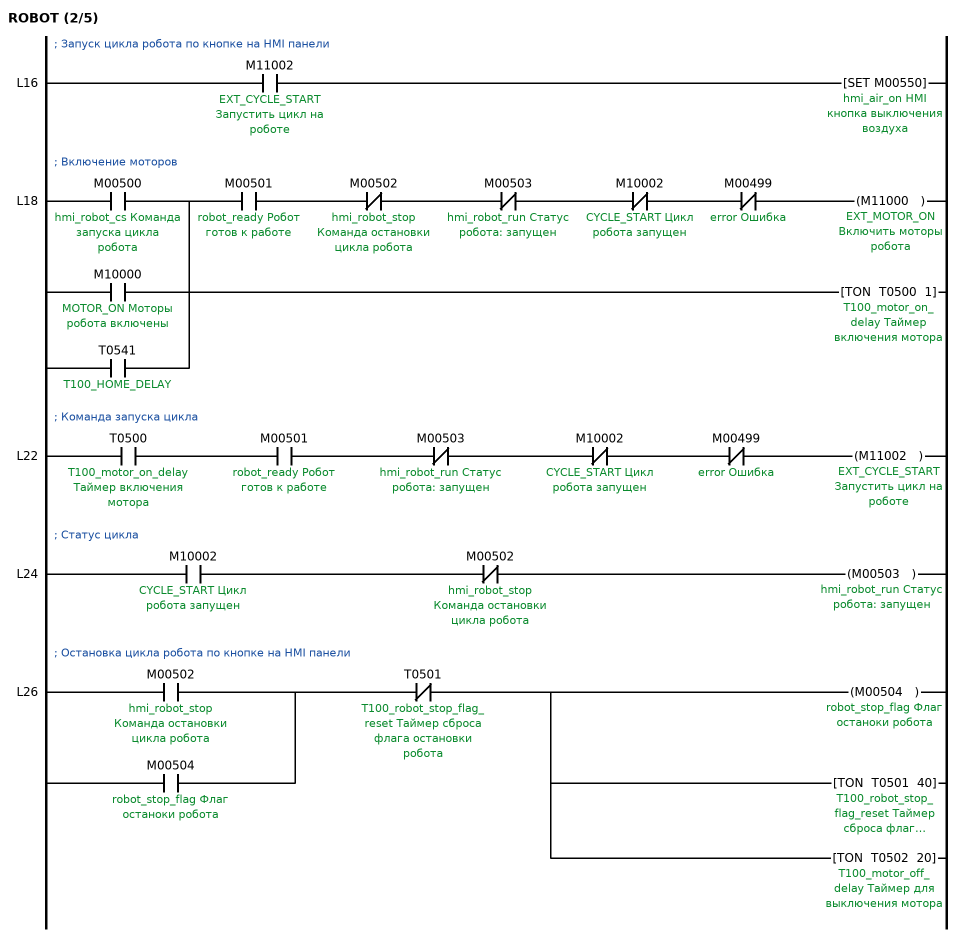
// Запуск цикла робота по кнопке на HMI панели
; L16
LOAD      M11002	// EXT_CYCLE_START Запустить цикл на роботе
SET       M00550	// hmi_air_on HMI кнопка выключения воздуха
// Включение моторов
; L18
LOAD      M00500	// hmi_robot_cs Команда запуска цикла робота
OR        M10000	// MOTOR_ON Моторы робота включены
OR        T0541	// T100_HOME_DELAY
MPUSH
AND       M00501	// robot_ready Робот готов к работе
AND NOT   M00502	// hmi_robot_stop Команда остановки цикла робота
AND NOT   M00503	// hmi_robot_run Статус робота: запущен
AND NOT   M10002	// CYCLE_START Цикл робота запущен
AND NOT   M00499	// error Ошибка
OUT       M11000	// EXT_MOTOR_ON Включить моторы робота
MPOP
TON       T0500 1	// T100_motor_on_delay Таймер включения мотора
// Команда запуска цикла
; L22
LOAD      T0500	// T100_motor_on_delay Таймер включения мотора
AND       M00501	// robot_ready Робот готов к работе
AND NOT   M00503	// hmi_robot_run Статус робота: запущен
AND NOT   M10002	// CYCLE_START Цикл робота запущен
AND NOT   M00499	// error Ошибка
OUT       M11002	// EXT_CYCLE_START Запустить цикл на роботе
// Статус цикла
; L24
LOAD      M10002	// CYCLE_START Цикл робота запущен
AND NOT   M00502	// hmi_robot_stop Команда остановки цикла робота
OUT       M00503	// hmi_robot_run Статус робота: запущен
// Остановка цикла робота по кнопке на HMI панели
; L26
LOAD      M00502	// hmi_robot_stop Команда остановки цикла робота
OR        M00504	// robot_stop_flag Флаг останоки робота
AND NOT   T0501	// T100_robot_stop_flag_reset Таймер сброса флага остановки робота
OUT       M00504	// robot_stop_flag Флаг останоки робота
TON       T0501 40	// T100_robot_stop_flag_reset Таймер сброса флага остановки робота
TON       T0502 20	// T100_motor_off_delay Таймер для выключения мотора

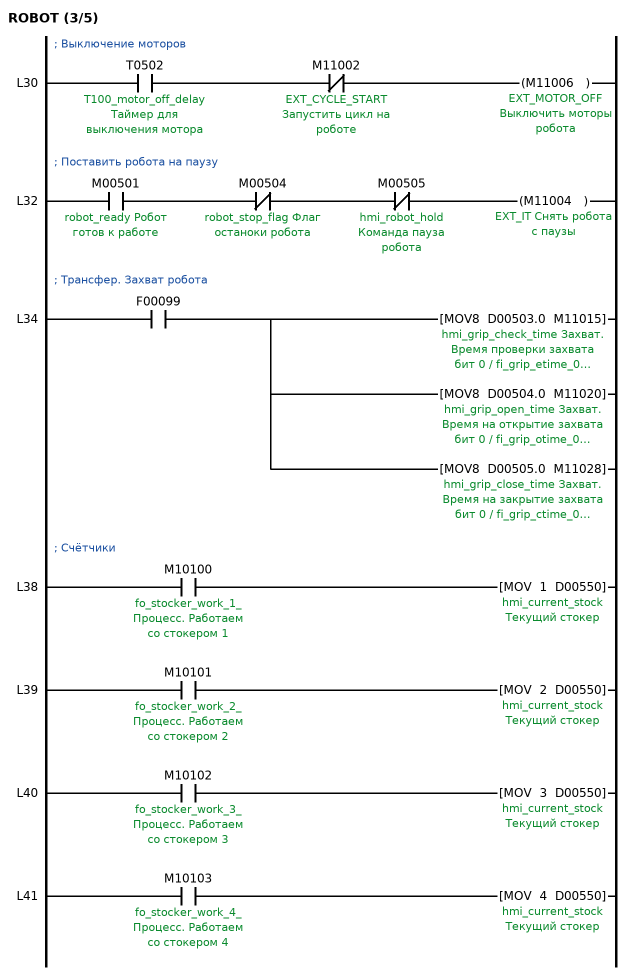
// Выключение моторов
; L30
LOAD      T0502	// T100_motor_off_delay Таймер для выключения мотора
AND NOT   M11002	// EXT_CYCLE_START Запустить цикл на роботе
OUT       M11006	// EXT_MOTOR_OFF Выключить моторы робота
// Поставить робота на паузу
; L32
LOAD      M00501	// robot_ready Робот готов к работе
AND NOT   M00504	// robot_stop_flag Флаг останоки робота
AND NOT   M00505	// hmi_robot_hold Команда пауза робота
OUT       M11004	// EXT_IT Снять робота с паузы
// Трансфер. Захват робота
; L34
LOAD      F00099
MOV8      D00503.0 M11015	// hmi_grip_check_time Захват. Время проверки захвата бит 0 / fi_grip_etime_0_ Захват. Время проверки захвата бит 0
MOV8      D00504.0 M11020	// hmi_grip_open_time Захват. Время на открытие захвата бит 0 / fi_grip_otime_0_ Захват. Время на открытие захвата бит 0
MOV8      D00505.0 M11028	// hmi_grip_close_time Захват. Время на закрытие захвата бит 0 / fi_grip_ctime_0_ Захват. Время на закрытие захвата бит 0
// Счётчики
; L38
LOAD      M10100	// fo_stocker_work_1_ Процесс. Работаем со стокером 1
MOV       1 D00550	// hmi_current_stock Текущий стокер
; L39
LOAD      M10101	// fo_stocker_work_2_ Процесс. Работаем со стокером 2
MOV       2 D00550	// hmi_current_stock Текущий стокер
; L40
LOAD      M10102	// fo_stocker_work_3_ Процесс. Работаем со стокером 3
MOV       3 D00550	// hmi_current_stock Текущий стокер
; L41
LOAD      M10103	// fo_stocker_work_4_ Процесс. Работаем со стокером 4
MOV       4 D00550	// hmi_current_stock Текущий стокер

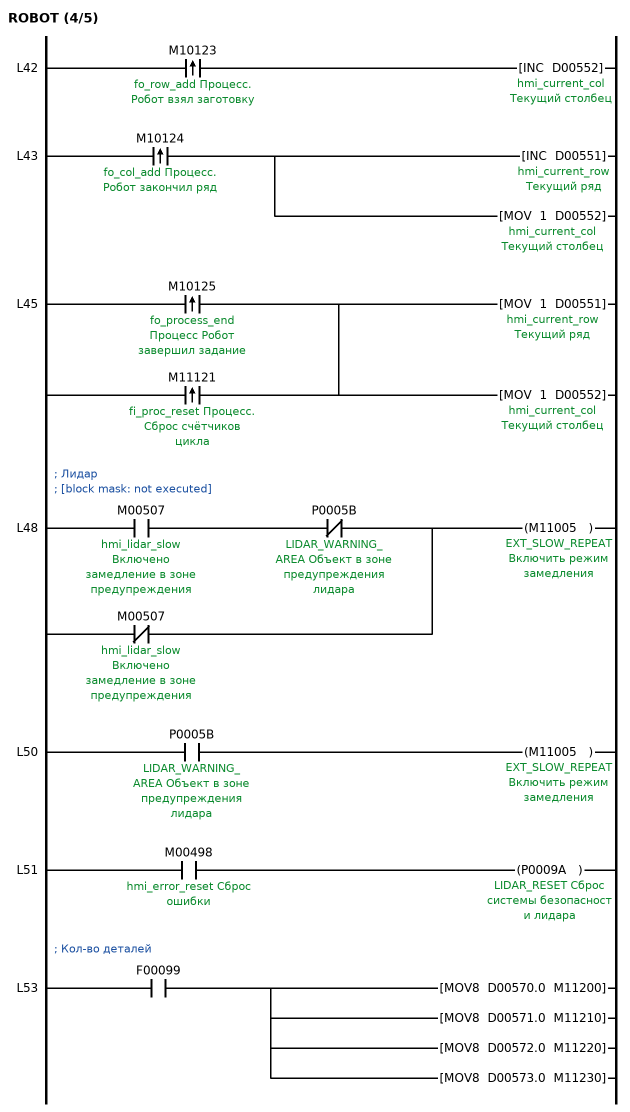
; L42
LOADP     M10123	// fo_row_add Процесс. Робот взял заготовку
INC       D00552	// hmi_current_col Текущий столбец
; L43
LOADP     M10124	// fo_col_add Процесс. Робот закончил ряд
INC       D00551	// hmi_current_row Текущий ряд
MOV       1 D00552	// hmi_current_col Текущий столбец
; L45
LOADP     M10125	// fo_process_end Процесс Робот завершил задание
ORP       M11121	// fi_proc_reset Процесс. Сброс счётчиков цикла
MOV       1 D00551	// hmi_current_row Текущий ряд
MOV       1 D00552	// hmi_current_col Текущий столбец
// Лидар
; L48 (block mask: not executed)
LOAD      M00507	// hmi_lidar_slow Включено замедление в зоне предупреждения
AND NOT   P0005B	// LIDAR_WARNING_AREA Объект в зоне предупреждения лидара
OR NOT    M00507	// hmi_lidar_slow Включено замедление в зоне предупреждения
OUT       M11005	// EXT_SLOW_REPEAT Включить режим замедления
; L50
LOAD      P0005B	// LIDAR_WARNING_AREA Объект в зоне предупреждения лидара
OUT       M11005	// EXT_SLOW_REPEAT Включить режим замедления
; L51
LOAD      M00498	// hmi_error_reset Сброс ошибки
OUT       P0009A	// LIDAR_RESET Сброс системы безопасности лидара
// Кол-во деталей
; L53
LOAD      F00099
MOV8      D00570.0 M11200
MOV8      D00571.0 M11210
MOV8      D00572.0 M11220
MOV8      D00573.0 M11230

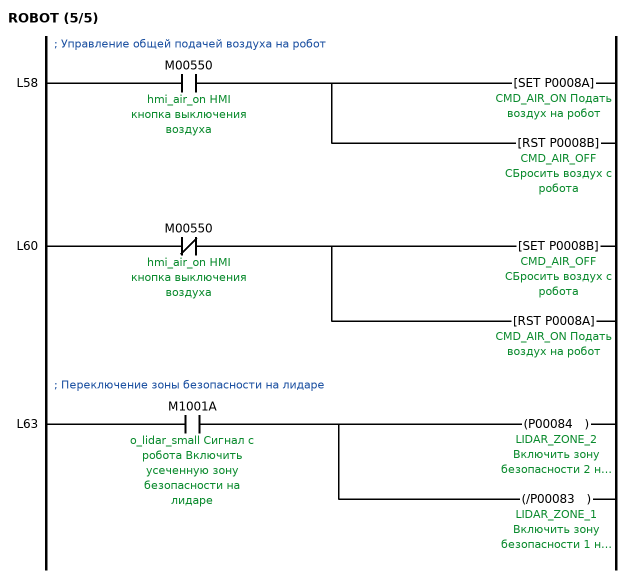
// Управление общей подачей воздуха на робот
; L58
LOAD      M00550	// hmi_air_on HMI кнопка выключения воздуха
SET       P0008A	// CMD_AIR_ON Подать воздух на робот
RST       P0008B	// CMD_AIR_OFF СБросить воздух с робота
; L60
LOAD NOT  M00550	// hmi_air_on HMI кнопка выключения воздуха
SET       P0008B	// CMD_AIR_OFF СБросить воздух с робота
RST       P0008A	// CMD_AIR_ON Подать воздух на робот
// Переключение зоны безопасности на лидаре
; L63
LOAD      M1001A	// o_lidar_small Сигнал с робота Включить усеченную зону безопасности на лидаре
OUT       P00084	// LIDAR_ZONE_2 Включить зону безопасности 2 на лидаре (усеченная)
OUT NOT   P00083	// LIDAR_ZONE_1 Включить зону безопасности 1 на лидаре (рабочая)

PROGRAM HMI (task: Scan Program)

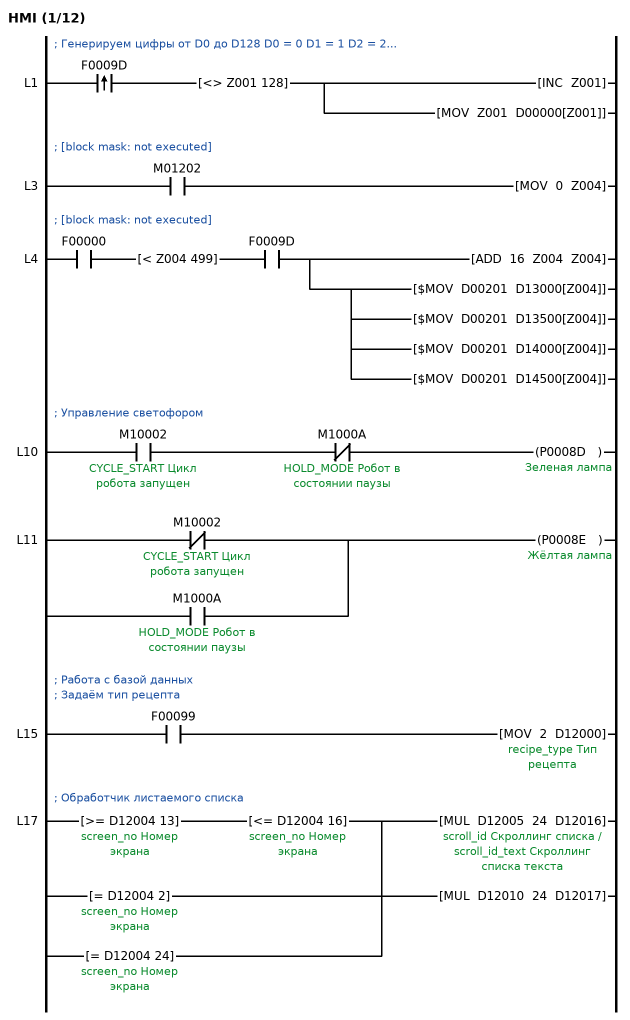
// Генерируем цифры от D0 до D128 D0 = 0 D1 = 1 D2 = 2...
; L1
LOADP     F0009D
AND<>     Z001 128
INC       Z001
MOV       Z001 D00000[Z001]
; L3 (block mask: not executed)
LOAD      M01202
MOV       0 Z004
; L4 (block mask: not executed)
LOAD      F00000
AND<      Z004 499
AND       F0009D
ADD       16 Z004 Z004
$MOV      D00201 D13000[Z004]
$MOV      D00201 D13500[Z004]
$MOV      D00201 D14000[Z004]
$MOV      D00201 D14500[Z004]
// Управление светофором
; L10
LOAD      M10002	// CYCLE_START Цикл робота запущен
AND NOT   M1000A	// HOLD_MODE Робот в состоянии паузы
OUT       P0008D	// Зеленая лампа
; L11
LOAD NOT  M10002	// CYCLE_START Цикл робота запущен
OR        M1000A	// HOLD_MODE Робот в состоянии паузы
OUT       P0008E	// Жёлтая лампа
// Работа с базой данных
// Задаём тип рецепта
; L15
LOAD      F00099
MOV       2 D12000	// recipe_type Тип рецепта
// Обработчик листаемого списка
; L17
LOAD>=    D12004 13	// screen_no Номер экрана
AND<=     D12004 16	// screen_no Номер экрана
OR=       D12004 2	// screen_no Номер экрана
OR=       D12004 24	// screen_no Номер экрана
MUL       D12005 24 D12016	// scroll_id Скроллинг списка / scroll_id_text Скроллинг списка текста
MUL       D12010 24 D12017

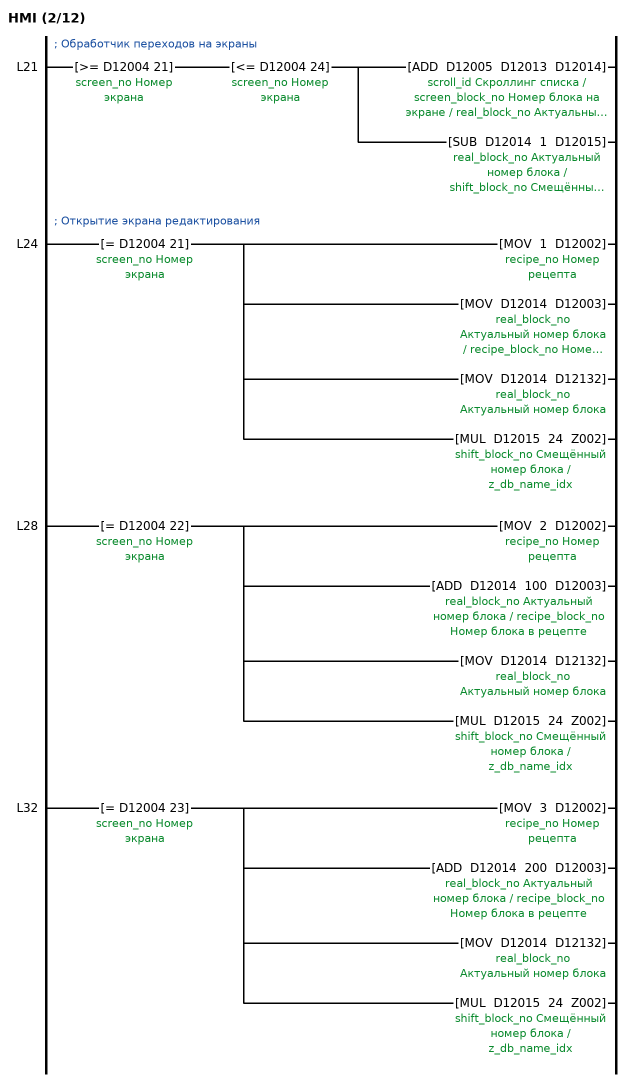
// Обработчик переходов на экраны
; L21
LOAD>=    D12004 21	// screen_no Номер экрана
AND<=     D12004 24	// screen_no Номер экрана
ADD       D12005 D12013 D12014	// scroll_id Скроллинг списка / screen_block_no Номер блока на экране / real_block_no Актуальный номер блока
SUB       D12014 1 D12015	// real_block_no Актуальный номер блока / shift_block_no Смещённый номер блока
// Открытие экрана редактирования
; L24
LOAD=     D12004 21	// screen_no Номер экрана
MOV       1 D12002	// recipe_no Номер рецепта
MOV       D12014 D12003	// real_block_no Актуальный номер блока / recipe_block_no Номер блока в рецепте
MOV       D12014 D12132	// real_block_no Актуальный номер блока
MUL       D12015 24 Z002	// shift_block_no Смещённый номер блока / z_db_name_idx
; L28
LOAD=     D12004 22	// screen_no Номер экрана
MOV       2 D12002	// recipe_no Номер рецепта
ADD       D12014 100 D12003	// real_block_no Актуальный номер блока / recipe_block_no Номер блока в рецепте
MOV       D12014 D12132	// real_block_no Актуальный номер блока
MUL       D12015 24 Z002	// shift_block_no Смещённый номер блока / z_db_name_idx
; L32
LOAD=     D12004 23	// screen_no Номер экрана
MOV       3 D12002	// recipe_no Номер рецепта
ADD       D12014 200 D12003	// real_block_no Актуальный номер блока / recipe_block_no Номер блока в рецепте
MOV       D12014 D12132	// real_block_no Актуальный номер блока
MUL       D12015 24 Z002	// shift_block_no Смещённый номер блока / z_db_name_idx

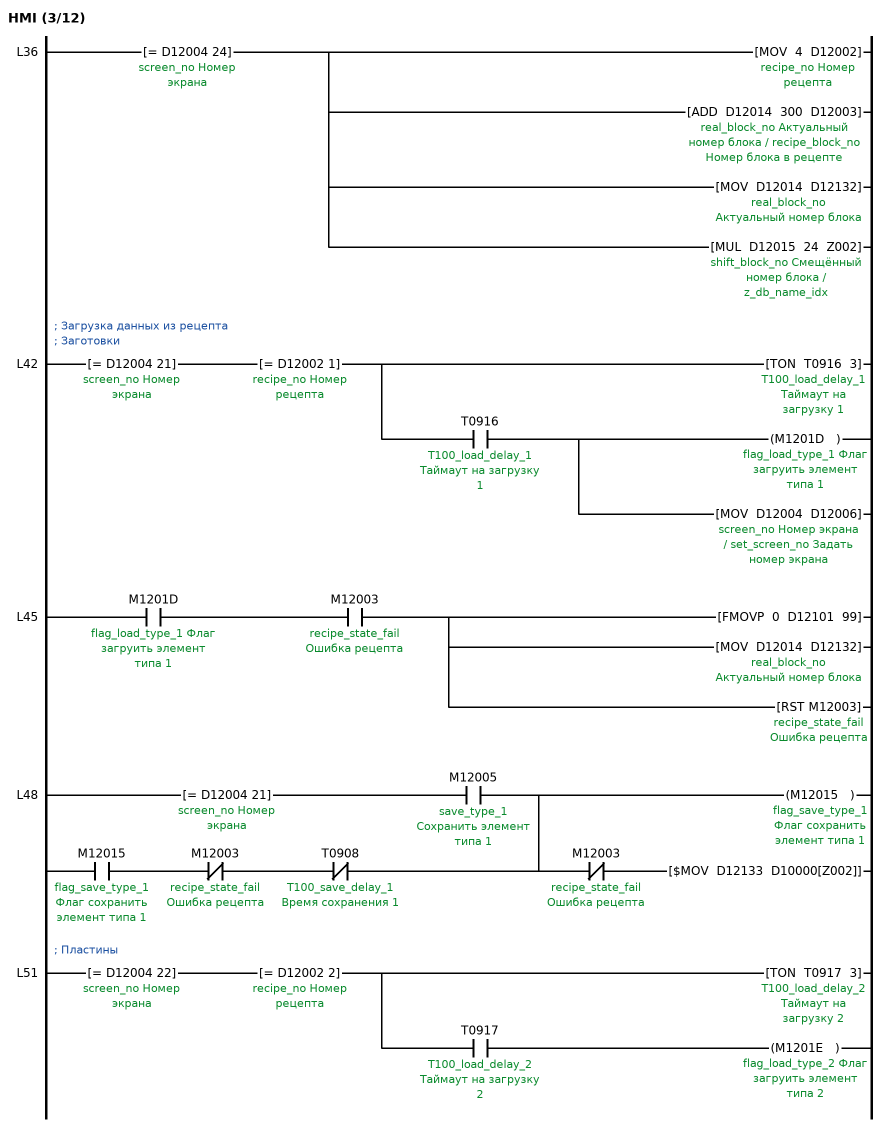
; L36
LOAD=     D12004 24	// screen_no Номер экрана
MOV       4 D12002	// recipe_no Номер рецепта
ADD       D12014 300 D12003	// real_block_no Актуальный номер блока / recipe_block_no Номер блока в рецепте
MOV       D12014 D12132	// real_block_no Актуальный номер блока
MUL       D12015 24 Z002	// shift_block_no Смещённый номер блока / z_db_name_idx
// Загрузка данных из рецепта
// Заготовки
; L42
LOAD=     D12004 21	// screen_no Номер экрана
AND=      D12002 1	// recipe_no Номер рецепта
TON       T0916 3	// T100_load_delay_1 Таймаут на загрузку 1
AND       T0916	// T100_load_delay_1 Таймаут на загрузку 1
OUT       M1201D	// flag_load_type_1 Флаг загруить элемент типа 1
MOV       D12004 D12006	// screen_no Номер экрана / set_screen_no Задать номер экрана
; L45
LOAD      M1201D	// flag_load_type_1 Флаг загруить элемент типа 1
AND       M12003	// recipe_state_fail Ошибка рецепта
FMOVP     0 D12101 99
MOV       D12014 D12132	// real_block_no Актуальный номер блока
RST       M12003	// recipe_state_fail Ошибка рецепта
; L48
LOAD=     D12004 21	// screen_no Номер экрана
AND       M12005	// save_type_1 Сохранить элемент типа 1
LOAD      M12015	// flag_save_type_1 Флаг сохранить элемент типа 1
AND NOT   M12003	// recipe_state_fail Ошибка рецепта
AND NOT   T0908	// T100_save_delay_1 Время сохранения 1
OR LOAD
OUT       M12015	// flag_save_type_1 Флаг сохранить элемент типа 1
AND NOT   M12003	// recipe_state_fail Ошибка рецепта
$MOV      D12133 D10000[Z002]
// Пластины
; L51
LOAD=     D12004 22	// screen_no Номер экрана
AND=      D12002 2	// recipe_no Номер рецепта
TON       T0917 3	// T100_load_delay_2 Таймаут на загрузку 2
AND       T0917	// T100_load_delay_2 Таймаут на загрузку 2
OUT       M1201E	// flag_load_type_2 Флаг загруить элемент типа 2

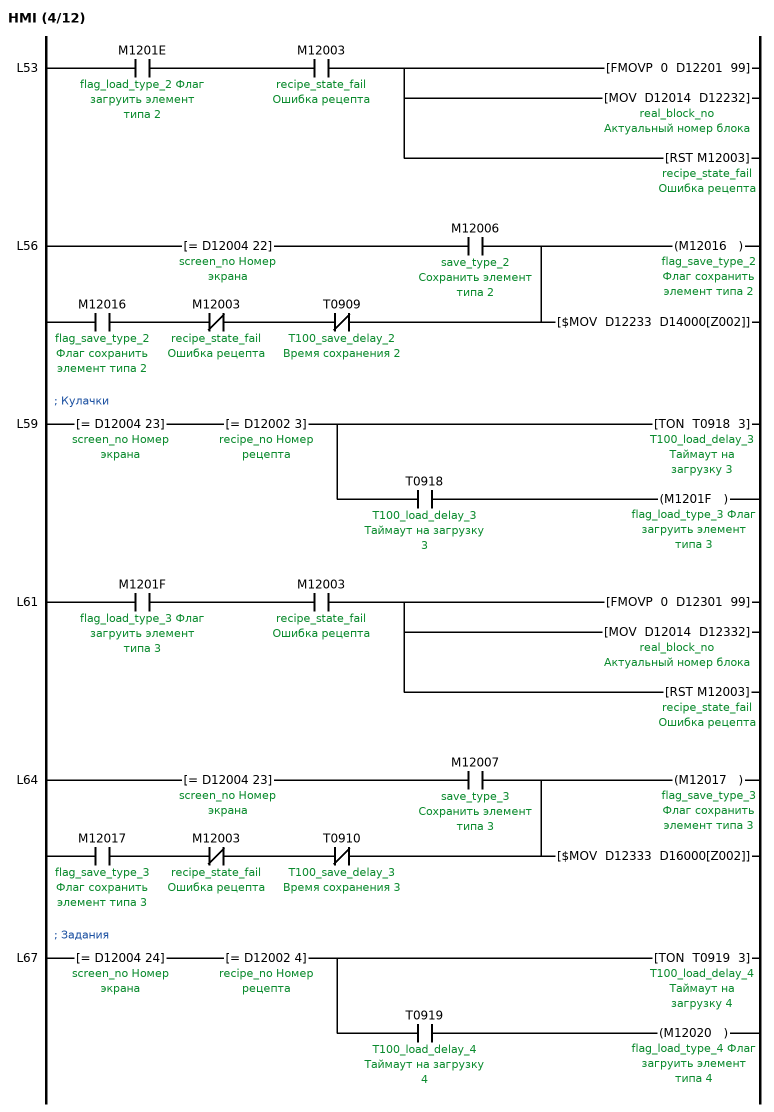
; L53
LOAD      M1201E	// flag_load_type_2 Флаг загруить элемент типа 2
AND       M12003	// recipe_state_fail Ошибка рецепта
FMOVP     0 D12201 99
MOV       D12014 D12232	// real_block_no Актуальный номер блока
RST       M12003	// recipe_state_fail Ошибка рецепта
; L56
LOAD=     D12004 22	// screen_no Номер экрана
AND       M12006	// save_type_2 Сохранить элемент типа 2
LOAD      M12016	// flag_save_type_2 Флаг сохранить элемент типа 2
AND NOT   M12003	// recipe_state_fail Ошибка рецепта
AND NOT   T0909	// T100_save_delay_2 Время сохранения 2
OR LOAD
OUT       M12016	// flag_save_type_2 Флаг сохранить элемент типа 2
$MOV      D12233 D14000[Z002]
// Кулачки
; L59
LOAD=     D12004 23	// screen_no Номер экрана
AND=      D12002 3	// recipe_no Номер рецепта
TON       T0918 3	// T100_load_delay_3 Таймаут на загрузку 3
AND       T0918	// T100_load_delay_3 Таймаут на загрузку 3
OUT       M1201F	// flag_load_type_3 Флаг загруить элемент типа 3
; L61
LOAD      M1201F	// flag_load_type_3 Флаг загруить элемент типа 3
AND       M12003	// recipe_state_fail Ошибка рецепта
FMOVP     0 D12301 99
MOV       D12014 D12332	// real_block_no Актуальный номер блока
RST       M12003	// recipe_state_fail Ошибка рецепта
; L64
LOAD=     D12004 23	// screen_no Номер экрана
AND       M12007	// save_type_3 Сохранить элемент типа 3
LOAD      M12017	// flag_save_type_3 Флаг сохранить элемент типа 3
AND NOT   M12003	// recipe_state_fail Ошибка рецепта
AND NOT   T0910	// T100_save_delay_3 Время сохранения 3
OR LOAD
OUT       M12017	// flag_save_type_3 Флаг сохранить элемент типа 3
$MOV      D12333 D16000[Z002]
// Задания
; L67
LOAD=     D12004 24	// screen_no Номер экрана
AND=      D12002 4	// recipe_no Номер рецепта
TON       T0919 3	// T100_load_delay_4 Таймаут на загрузку 4
AND       T0919	// T100_load_delay_4 Таймаут на загрузку 4
OUT       M12020	// flag_load_type_4 Флаг загруить элемент типа 4

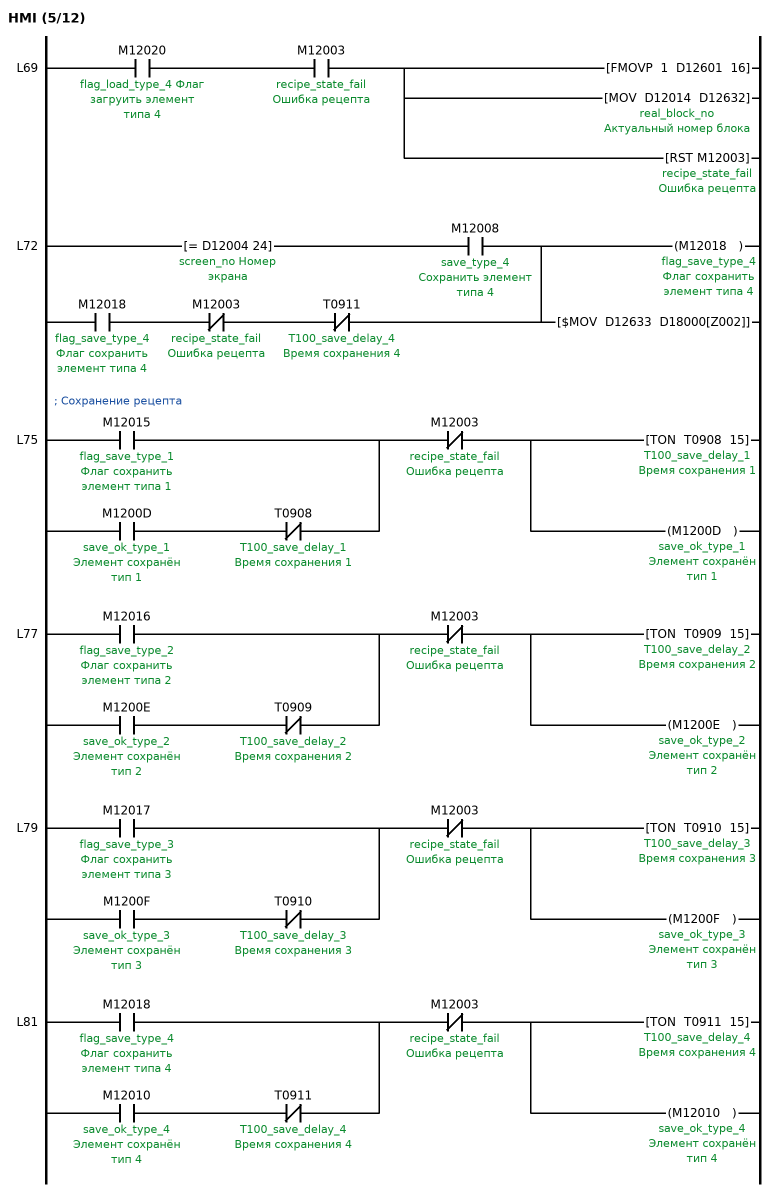
; L69
LOAD      M12020	// flag_load_type_4 Флаг загруить элемент типа 4
AND       M12003	// recipe_state_fail Ошибка рецепта
FMOVP     1 D12601 16
MOV       D12014 D12632	// real_block_no Актуальный номер блока
RST       M12003	// recipe_state_fail Ошибка рецепта
; L72
LOAD=     D12004 24	// screen_no Номер экрана
AND       M12008	// save_type_4 Сохранить элемент типа 4
LOAD      M12018	// flag_save_type_4 Флаг сохранить элемент типа 4
AND NOT   M12003	// recipe_state_fail Ошибка рецепта
AND NOT   T0911	// T100_save_delay_4 Время сохранения 4
OR LOAD
OUT       M12018	// flag_save_type_4 Флаг сохранить элемент типа 4
$MOV      D12633 D18000[Z002]
// Сохранение рецепта
; L75
LOAD      M12015	// flag_save_type_1 Флаг сохранить элемент типа 1
LOAD      M1200D	// save_ok_type_1 Элемент сохранён тип 1
AND NOT   T0908	// T100_save_delay_1 Время сохранения 1
OR LOAD
AND NOT   M12003	// recipe_state_fail Ошибка рецепта
TON       T0908 15	// T100_save_delay_1 Время сохранения 1
OUT       M1200D	// save_ok_type_1 Элемент сохранён тип 1
; L77
LOAD      M12016	// flag_save_type_2 Флаг сохранить элемент типа 2
LOAD      M1200E	// save_ok_type_2 Элемент сохранён тип 2
AND NOT   T0909	// T100_save_delay_2 Время сохранения 2
OR LOAD
AND NOT   M12003	// recipe_state_fail Ошибка рецепта
TON       T0909 15	// T100_save_delay_2 Время сохранения 2
OUT       M1200E	// save_ok_type_2 Элемент сохранён тип 2
; L79
LOAD      M12017	// flag_save_type_3 Флаг сохранить элемент типа 3
LOAD      M1200F	// save_ok_type_3 Элемент сохранён тип 3
AND NOT   T0910	// T100_save_delay_3 Время сохранения 3
OR LOAD
AND NOT   M12003	// recipe_state_fail Ошибка рецепта
TON       T0910 15	// T100_save_delay_3 Время сохранения 3
OUT       M1200F	// save_ok_type_3 Элемент сохранён тип 3
; L81
LOAD      M12018	// flag_save_type_4 Флаг сохранить элемент типа 4
LOAD      M12010	// save_ok_type_4 Элемент сохранён тип 4
AND NOT   T0911	// T100_save_delay_4 Время сохранения 4
OR LOAD
AND NOT   M12003	// recipe_state_fail Ошибка рецепта
TON       T0911 15	// T100_save_delay_4 Время сохранения 4
OUT       M12010	// save_ok_type_4 Элемент сохранён тип 4

